TYPE "PLCtoMES_ST350_ext"
VERSION : 0.1
   STRUCT
      MainCheckIn : "PLCtoMES_MainCheckIn_ext";
      SubCheckIn : "PLCtoMES_SubCheckIn_ext";
      ScanResultsStored : "PLCtoMES_ResultsStoredScanExchange_ext";
      PrintExchange : "PLCtoMES_PrintExchange_ext";
      MainCheckOut : "PLCtoMES_MainCheckOut_ext";
      Common : "PLCtoMES_Common_ext";
   END_STRUCT;

END_TYPE

